TYPE ST_CTRL_TRIGGER :
STRUCT
  Control             : T_TriggerControlBits;

   {attribute 'hide'}
  byc : ARRAY[1..7] OF BYTE;;


  AxisId              : UDINT;  // TwinCAT NC Axis ID

  TriggerCount        : UDINT;  // how many TriggerPositions shall be used

  TriggerPosition     : ARRAY[1..MAX_TRIGGER_COUNT] OF LREAL;  // Axis Position where output must be set by TriggerBox
                                // Trigger is set when crossing Position
END_STRUCT
END_TYPE

(* stored: Version 1.1.0.1, ProductVersion 3.1.4024.13
   DUT ST_CTRL_TRIGGER: Id {1c130404-c118-4db3-a522-21c1b1383288} *)
